% RSLogix 500 project MALETA_BAK059.RSS %
PROJECT "UNTITLED"    % processor: MicroLogix 1200 %

PROGRAM FILES
  LAD 2   10 rungs
  LAD 3   12 rungs

DATA FILES
  O0 OUTPUT  6 elements
  I1 INPUT  10 elements
  S2 STATUS  66 elements
  B3 BINARY  1 elements
  T4 TIMER  1 elements
  C5 COUNTER  1 elements
  R6 CONTROL  1 elements
  N7 INTEGER  1 elements

LADDER 2
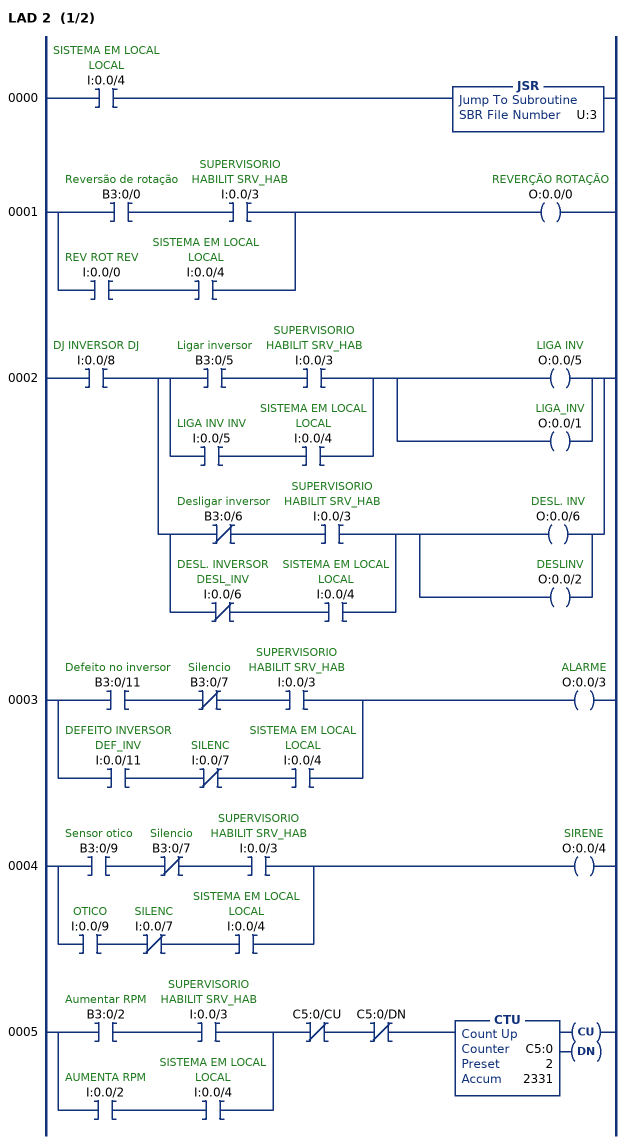
% Rung: 0 %
SOR XIC I:0.0/4 JSR U:3 EOR
%   I:0.0/4  LOCAL  "SISTEMA EM LOCAL" %
% Rung: 1 %
SOR BST XIC B3:0/0 XIC I:0.0/3 NXB XIC I:0.0/0 XIC I:0.0/4 BND OTE O:0.0/0 EOR
%   B3:0/0  "Reversão de rotação" %
%   I:0.0/3  SRV_HAB  "SUPERVISORIO HABILIT" %
%   I:0.0/0  REV  "REV ROT" %
%   I:0.0/4  LOCAL  "SISTEMA EM LOCAL" %
%   O:0.0/0  "REVERÇÃO ROTAÇÃO" %
% Rung: 2 %
SOR XIC I:0.0/8 BST BST XIC B3:0/5 XIC I:0.0/3 NXB XIC I:0.0/5 XIC I:0.0/4 BND BST OTE O:0.0/5 NXB OTE O:0.0/1 BND NXB BST XIO B3:0/6 XIC I:0.0/3 NXB XIO I:0.0/6 XIC I:0.0/4 BND BST OTE O:0.0/6 NXB OTE O:0.0/2 BND BND EOR
%   I:0.0/8  DJ  "DJ INVERSOR" %
%   B3:0/5  "Ligar inversor" %
%   I:0.0/3  SRV_HAB  "SUPERVISORIO HABILIT" %
%   I:0.0/5  INV  "LIGA INV" %
%   I:0.0/4  LOCAL  "SISTEMA EM LOCAL" %
%   O:0.0/5  "LIGA INV" %
%   O:0.0/1  LIGA_INV %
%   B3:0/6  "Desligar inversor" %
%   I:0.0/6  DESL_INV  "DESL. INVERSOR" %
%   O:0.0/6  "DESL. INV" %
%   O:0.0/2  DESLINV %
% Rung: 3 %
SOR BST XIC B3:0/11 XIO B3:0/7 XIC I:0.0/3 NXB XIC I:0.0/11 XIO I:0.0/7 XIC I:0.0/4 BND OTE O:0.0/3 EOR
%   B3:0/11  "Defeito no inversor" %
%   B3:0/7  "Silencio" %
%   I:0.0/3  SRV_HAB  "SUPERVISORIO HABILIT" %
%   I:0.0/11  DEF_INV  "DEFEITO INVERSOR" %
%   I:0.0/7  SILENC %
%   I:0.0/4  LOCAL  "SISTEMA EM LOCAL" %
%   O:0.0/3  ALARME %
% Rung: 4 %
SOR BST XIC B3:0/9 XIO B3:0/7 XIC I:0.0/3 NXB XIC I:0.0/9 XIO I:0.0/7 XIC I:0.0/4 BND OTE O:0.0/4 EOR
%   B3:0/9  "Sensor otico" %
%   B3:0/7  "Silencio" %
%   I:0.0/3  SRV_HAB  "SUPERVISORIO HABILIT" %
%   I:0.0/9  OTICO %
%   I:0.0/7  SILENC %
%   I:0.0/4  LOCAL  "SISTEMA EM LOCAL" %
%   O:0.0/4  SIRENE %
% Rung: 5 %
SOR BST XIC B3:0/2 XIC I:0.0/3 NXB XIC I:0.0/2 XIC I:0.0/4 BND XIO C5:0/CU XIO C5:0/DN CTU C5:0 2 2331 EOR
%   B3:0/2  "Aumentar RPM" %
%   I:0.0/3  SRV_HAB  "SUPERVISORIO HABILIT" %
%   I:0.0/2  "AUMENTA RPM" %
%   I:0.0/4  LOCAL  "SISTEMA EM LOCAL" %

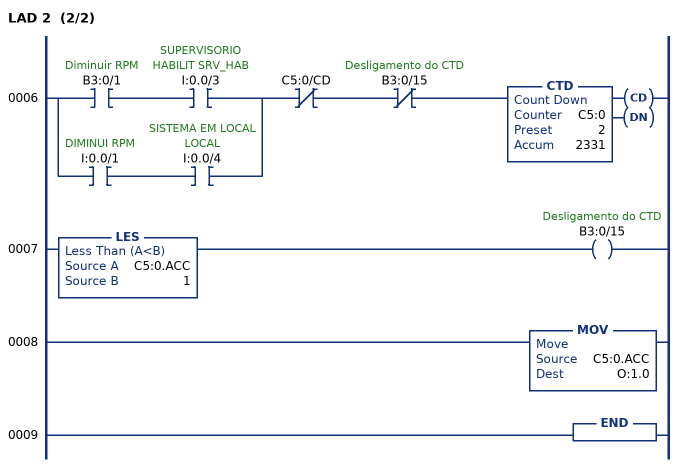
% Rung: 6 %
SOR BST XIC B3:0/1 XIC I:0.0/3 NXB XIC I:0.0/1 XIC I:0.0/4 BND XIO C5:0/CD XIO B3:0/15 CTD C5:0 2 2331 EOR
%   B3:0/1  "Diminuir RPM" %
%   I:0.0/3  SRV_HAB  "SUPERVISORIO HABILIT" %
%   I:0.0/1  "DIMINUI RPM" %
%   I:0.0/4  LOCAL  "SISTEMA EM LOCAL" %
%   B3:0/15  "Desligamento do CTD" %
% Rung: 7 %
SOR LES C5:0.ACC 1 OTE B3:0/15 EOR
%   B3:0/15  "Desligamento do CTD" %
% Rung: 8 %
SOR MOV C5:0.ACC O:1.0 EOR
% Rung: 9 %
SOR END EOR

LADDER 3
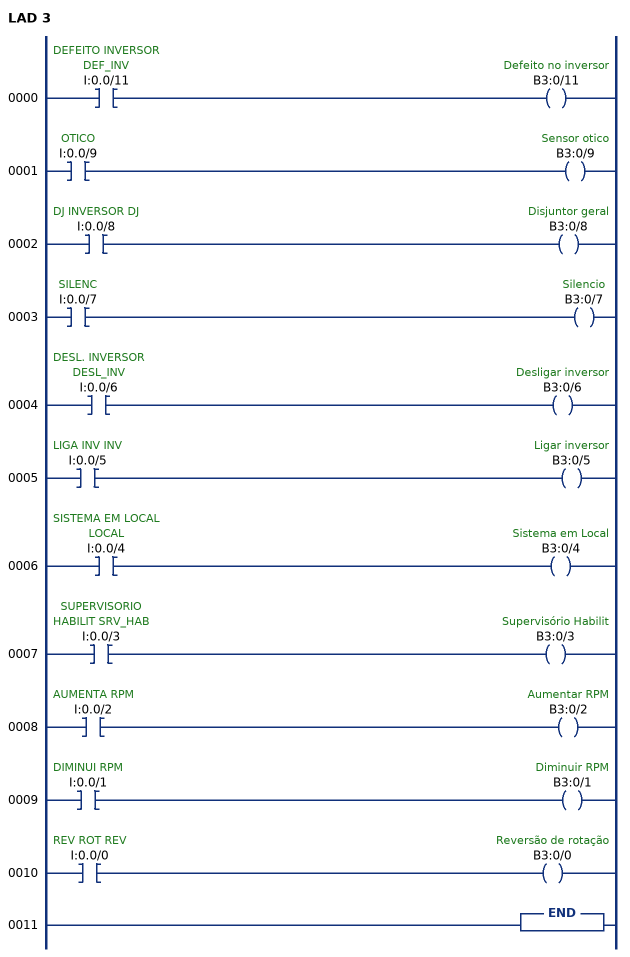
% Rung: 0 %
SOR XIC I:0.0/11 OTE B3:0/11 EOR
%   I:0.0/11  DEF_INV  "DEFEITO INVERSOR" %
%   B3:0/11  "Defeito no inversor" %
% Rung: 1 %
SOR XIC I:0.0/9 OTE B3:0/9 EOR
%   I:0.0/9  OTICO %
%   B3:0/9  "Sensor otico" %
% Rung: 2 %
SOR XIC I:0.0/8 OTE B3:0/8 EOR
%   I:0.0/8  DJ  "DJ INVERSOR" %
%   B3:0/8  "Disjuntor geral" %
% Rung: 3 %
SOR XIC I:0.0/7 OTE B3:0/7 EOR
%   I:0.0/7  SILENC %
%   B3:0/7  "Silencio" %
% Rung: 4 %
SOR XIC I:0.0/6 OTE B3:0/6 EOR
%   I:0.0/6  DESL_INV  "DESL. INVERSOR" %
%   B3:0/6  "Desligar inversor" %
% Rung: 5 %
SOR XIC I:0.0/5 OTE B3:0/5 EOR
%   I:0.0/5  INV  "LIGA INV" %
%   B3:0/5  "Ligar inversor" %
% Rung: 6 %
SOR XIC I:0.0/4 OTE B3:0/4 EOR
%   I:0.0/4  LOCAL  "SISTEMA EM LOCAL" %
%   B3:0/4  "Sistema em Local" %
% Rung: 7 %
SOR XIC I:0.0/3 OTE B3:0/3 EOR
%   I:0.0/3  SRV_HAB  "SUPERVISORIO HABILIT" %
%   B3:0/3  "Supervisório Habilit" %
% Rung: 8 %
SOR XIC I:0.0/2 OTE B3:0/2 EOR
%   I:0.0/2  "AUMENTA RPM" %
%   B3:0/2  "Aumentar RPM" %
% Rung: 9 %
SOR XIC I:0.0/1 OTE B3:0/1 EOR
%   I:0.0/1  "DIMINUI RPM" %
%   B3:0/1  "Diminuir RPM" %
% Rung: 10 %
SOR XIC I:0.0/0 OTE B3:0/0 EOR
%   I:0.0/0  REV  "REV ROT" %
%   B3:0/0  "Reversão de rotação" %
% Rung: 11 %
SOR END EOR

DATA TABLE (non-zero values as saved)
DATA B3
% B3:0 % 0X0009
DATA C5
% .PRE .ACC %
% C5:0 % 2 2331
